(* PLC project poST.project, poSTIDE *)
(* stored: creationDateTime 2021-08-31T00:00:00.000000 *)

FUNCTION SUB_DATE_DATE : TIME
  VAR_INPUT
    in1 : DATE;
    in2 : DATE;
  END_VAR

END_FUNCTION
